(* CODESYS project safetymonitoring.library
   Author: Adam Garner
   Placeholder: SafetyMonitoring
   Title: SafetyMonitoring
   Version: 0.1.0.0
   Company: Ljmu

Project tree, tasks and I/O mapping:
  libraries: Tc2_Standard, * (Beckhoff Automation GmbH); Tc2_System, * (Beckhoff Automation GmbH); Tc3_Module, * (Beckhoff Automation GmbH)
  DUTs/
    data type e_EstopFBState
    data type e_EthercatCommError
    data type e_EthercatError
    data type e_EthercatState
    data type e_SafetyDiag
    data type e_SafetyGroupDiagnosis
    data type e_SafetyGroupState
    data type e_SafetyState
    data type ST_EL1918Inputs
    data type ST_EL1957Inputs
    data type ST_EL1957Outputs
    data type ST_EL2904Outputs
    data type ST_EstopFB
    data type ST_EstopFBDiag
    data type ST_EthercatStatus
    data type St_ModuleDescription
    data type ST_SafetyModule
    data type ST_SafetyStatus
    data type ST_WcStateStandard
  GVLs/
  POUs/
    function F_EthercatStateValid [ST]
    function block FB_EL1918Monitor [ST]: FB_init, GetInputs, SetInputs
    function block FB_EL1957Monitor [ST]
    function block FB_EL2904Monitor [ST]: FB_init
    function block FB_EstopFBCollectors [ST]: GetEstopData, MasterDataValid
    function block FB_EthercatModuleMonitor [ST]: CreateEthercatStatus, EtherCatStatusValid, FB_init, GetEthercatStatus, GetModuleDescription, LinkedOkVaild, ModuleDataValid, SetEthercatInputs, SetModuleDescription
    function block FB_SafetyEstopMonitor [ST]: FB_init, GetEstopName, GetEstopState, GetFlags, GetState, Reset, SetState
    function block FB_SafetyModuleCollector [ST]: GetSafetyStatus
    function block FB_SafetyModuleMonitor [ST]: CreateSafetyStatus, FB_init, GetSafetyStatus, SetSafetyInputs, ValidateSafetyStatus
    function block FB_SafetySystemMonitor [ST]: GetGlobalEstopStatus, SetMasterStatus
    interface ITF_SafetyModuleMonitor: CreateSafetyStatus, FB_init, GetEthercatStatus, GetModuleDescription, GetSafetyStatus, SetEthercatInputs, SetSafetyInputs, ValidateSafetyStatus
    program MAIN [ST]
  VISUs/
*)

// DUTs/e_EstopFBState
{attribute 'qualified_only'}
{attribute 'to_string'}
// Enum decribes states of a Estop function block 
TYPE e_EstopFBState :
(
	Undefined := 0,
	Run :=1,
	Stop:=2,
	Safe:=3,
	Error:=4,
	Reset:=5,
	Start:=6,
	Delayout:=8 
)BYTE;
END_TYPE
//source https://www.beckhoff.com/media/downloads/downloads/twinsafe-logic-fb-3.pdf PG50

// DUTs/e_EthercatCommError
{attribute 'qualified_only'}
{attribute 'to_string'}

TYPE e_EthercatCommError :
(	NoError:=0,
	InvalidError:=1,
	CommPortA := 16#1000,
	CommPortB := 16#2000,
	CommPortC := 16#4000,
	CommPortD := 16#8000
	
)UINT;
END_TYPE
// source https://infosys.beckhoff.com/english.php?content=../content/1033/b110_ethercat_optioninterface/1976021643.html&id=

// DUTs/e_EthercatError
{attribute 'qualified_only'}
{attribute 'to_string'}
// errors on a ethercat module 
TYPE e_EthercatError :
(
	NoError:=16#0000,
	SlaveSignalsError := 16#0010,
	InvalidProductCode := 16#0020,
	InitError := 16#0040,
	SlaveDisabled:= 16#0080,
	SlaveNotPresent :=16#0100,
	SlaveSignalLinkError := 16#0200,
	SlaveSignalMissingLink := 16#0400,
	SlaveSignalsUnexpectedLink := 16#0800,
	InvalidError:=5
	
)UINT;
END_TYPE
//source https://infosys.beckhoff.com/english.php?content=../content/1033/b110_ethercat_optioninterface/1976021643.html&id=

// DUTs/e_EthercatState
{attribute 'qualified_only'}
{attribute 'to_string'}
// the states of any ethercat module can be in 
TYPE e_EthercatState :
(
	InvalidState:=0,
	INIT := 1,
	PREOP :=2,
	BOOT :=3,
	SAFEOP:=4,
	OP :=8

)BYTE;
END_TYPE

//source https://infosys.beckhoff.com/english.php?content=../content/1033/b110_ethercat_optioninterface/1976021643.html&id=

// DUTs/e_SafetyDiag
{attribute 'qualified_only'}
{attribute 'to_string'}
//Enum descibes the final 4 bits of the Diagnostic varible that is common to all twinsafe modules 
TYPE e_SafetyDiag :
(	NoDiagnosisData:=0,
	InvalidCommand := 2#01,
	UnknownCommand := 2#10,
	InvalidConnectionID := 2#11,
	InvalidCRC := 2#100,
	WatchdogElapsed := 2#101,
	InvalidFSoEAddr := 2#110,
	InvalidData := 2#111,
	InvalidCommsParameterLength := 2#1000,
	InvalidCommsParameters := 2#1001,
	InvalidUserParametersLength := 2#1010,
	InvalidUserParameters := 2#1011,
	FSoEMasterReset := 2#1100,
	ModuleErrorOnSlaveComErrorActive := 2#1101,
	ModuleErrorOnSlaveErrAckActive := 2#1110,
	SlaveNotStartedOrUnexpectedErrorArgument :=2#1111
	
	
)USINT;
END_TYPE
// source https://download.beckhoff.com/download/Document/automation/twinsafe/TwinSAFE-Logic-FBen.pdf pg 20

// DUTs/e_SafetyGroupDiagnosis
{attribute 'qualified_only'}
TYPE e_SafetyGroupDiagnosis :
(
	NoError := 0,
	FBError:=1, 		//at least one FB is in ERROR state 
	ComError:=2, 		// at least one connection is faulty 
	ModuleError:=3, 	//the input ModuleFault is 1 
	CmpError:=4, 		//On startup, at least one analog FB input deviates from the last saved value (Power-On Analog Value Check Error) 
	DeativateError:=5, 	//The timeout has elapsed while waiting for the COM error in "passivate" mode of a manual control unit 
	RestartError :=6    //The TwinSAFE logic program was restarted because the EtherCAT connection was restarted or a user logged in without 
						//reloading the TwinSAFE logic program (or parts of it).
	
)USINT
;
END_TYPE
 // https://www.beckhoff.com/media/downloads/downloads/twinsafe-logic-fb-3.pdf pg 26

// DUTs/e_SafetyGroupState
{attribute 'qualified_only'}
TYPE e_SafetyGroupState :
(
	InvalidState:=0,
	Run:=1,				//Input RUN=1, no error in the group, and all connections have started up without error
	Stop:=2,			//Input RUN = 0 
	Error:=4,			//Group is in error, see Diagnostic information 
	Reset:=5,			//After a group error has occurred, all errors have been rectified and the Err Ack signal is 1 
	Start:=6,			// The group remains in this state as long as not all connections have started up after the start of the group (RUN=1) 
	StopError:=7,		// When the group is started or initialized, it assumes the STOPERROR status if the TwinSAFE connections are assigned to the group. 
						//The group switches from STOPERROR state into ERROR state if the Run input is TRUE. 
	Deactive:=16, 		//Group was deactivated via customizing
	WaitComError:=17 	// This state is set when the customizing function "Passivate" is selected and the system waits for ComError of the group
	
	
)USINT
;
END_TYPE
// source https://www.beckhoff.com/media/downloads/downloads/twinsafe-logic-fb-3.pdf pg26

// DUTs/e_SafetyState
{attribute 'qualified_only'}
{attribute 'to_string'}
//Enum descibes the State varible that is common to all twinsafe modules 
TYPE e_SafetyState :
(
	Reset := 100,
	Session:=101,
	Connection:=102,
	Parameter:=103,
	Data:=104,
	Shutdown:=105,
	ShutDownDeactivate:=106,
	StateDataNotAvailable:=0,
	InvalidState :=1
)USINT :=InvalidState
;
END_TYPE
// source https://download.beckhoff.com/download/Document/automation/twinsafe/TwinSAFE-Logic-FBen.pdf pg 21

// DUTs/ST_EL1918Inputs
// bit structure showing raw input state of a EL1918 module (8 channel safe inputs) should be mapped to the IO module 
TYPE ST_EL1918Inputs :
STRUCT
	Input1 :BIT;
	Input1Err :BIT;
	Input2 :BIT;
	Input2Err :BIT;
	Input3 :BIT;
	Input3Err :BIT;
	Input4 :BIT;
	Input4Err :BIT;
	Input5 :BIT;
	Input5Err :BIT;
	Input6 :BIT;
	Input6Err :BIT;
	Input7 :BIT;
	Input7Err :BIT;
	Input8 :BIT;
	Input8Err :BIT;
END_STRUCT
END_TYPE

// DUTs/ST_EL1957Inputs
// bit structure for all inputs of a E1957 8 channel safe input 4 safe outputs should be mapped to the IO 
TYPE ST_EL1957Inputs :
STRUCT
	Output1Err :BIT;// True if output 1 is in error state 
	Output2Err :BIT;
	Output3Err :BIT;
	Output4Err :BIT;
	Input1 :BIT;
	Input2 :BIT;
	Module1Err :BIT;//module 1 contains inputs 1 & 2 
	Input3 :BIT;
	Input4 :BIT;
	Module2Err :BIT;//module 2 contains inputs 3 & 4
	Input5 :BIT;
	Input6 :BIT;
	Module3Err :BIT;//module 3 contains inputs 5 & 6
	Input7 :BIT;
	Input8 :BIT;
	Module4Err :BIT;//module 4 contains inputs 7 & 8 
END_STRUCT
END_TYPE

// DUTs/ST_EL1957Outputs
TYPE ST_EL1957Outputs :
STRUCT
	Output1 :BIT;
	Output1ErrAck :BIT;
	Output2 :BIT;
	Output2ErrAck :BIT;
	Output3 :BIT;
	Output3ErrAck :BIT;
	Output4 :BIT;
	Output4ErrAck :BIT;
	InputModule1ErrAck :BIT;
	InputModule2ErrAck :BIT;
	InputModule3ErrAck :BIT;
	InputModule4ErrAck :BIT;
	
END_STRUCT
END_TYPE

// DUTs/ST_EL2904Outputs
TYPE ST_EL2904Outputs :
STRUCT
	Output1 :BIT;
	Output2 :BIT;
	Output3 :BIT;
	Output4 :BIT;
END_STRUCT
END_TYPE

// DUTs/ST_EstopFB
TYPE ST_EstopFB :
STRUCT
	EstopArea :STRING;
	State : e_EstopFBState;
	StrState: STRING;
	Diagnostics : ST_EstopFBDiag;
	Running :BOOL;
	Error:BOOL;
	Restart :BOOL;
END_STRUCT
END_TYPE

// DUTs/ST_EstopFBDiag
TYPE ST_EstopFBDiag :
STRUCT
	DiscrepancyErrInputGroup1 :BIT;
	DiscrepancyErrInputGroup2 :BIT;
	DiscrepancyErrInputGroup3 :BIT;
	DiscrepancyErrInputGroup4 :BIT;
	EDM1Err :BIT;
	EDM2Err :BIT;
	NA_1 :BIT;
	NA_2 :BIT;
	DiscErrInputGroup1 :BIT;
	DiscErrInputGroup2 :BIT;
	DiscErrInputGroup3 :BIT;
	DiscErrInputGroup4 :BIT;
	NA_3 :BIT;
	NA_4: BIT;
	NA_5: BIT;
	NA_6: BIT;
END_STRUCT
END_TYPE
// source https://www.beckhoff.com/media/downloads/downloads/twinsafe-logic-fb-3.pdf pg47

// DUTs/ST_EthercatStatus
// readable structure showing the status of any ethercat module 
TYPE ST_EthercatStatus :
STRUCT
	State :e_EthercatState;
	Error :e_EthercatError;
	CommError :e_EthercatCommError;
	DataValid:BOOL; // if false all data values from the module arent current 
	CablesOk:BOOL; // true if no comms error showing 
	LinkedOK :BOOL; // true if the values are linked to a module 
	ModuleOK:BOOL; // true is all values are normal excluding cables ok 
END_STRUCT
END_TYPE


// ethercat state definition https://infosys.beckhoff.com/english.php?content=../content/1033/tcsystemmanager/1089009035.html&id=4933952924797561914

// DUTs/St_ModuleDescription

//structure for storing data about the modules that are being monitored
TYPE St_ModuleDescription :
STRUCT
	ModuleName: STRING; // related to that it does 
	ModuleElectricalRef :STRING; // as shown on the wiring diagram
	ModuleAddress : INT; // termingal number shown in twincat 
	
END_STRUCT
END_TYPE

// DUTs/ST_SafetyModule
TYPE ST_SafetyModule :
STRUCT
	SafetyStatus : ST_SafetyStatus;
	strSafetyState :STRING;
	strSafetydiag :STRING;
	EthercatStatus : ST_EthercatStatus;
	strEthercatState : STRING;
	strEthercatError : STRING;
	strEthercatCommError : STRING;
	ModuleDescription : St_ModuleDescription; 
END_STRUCT
END_TYPE

// DUTs/ST_SafetyStatus
// readable structure for the current status of a safety module 
TYPE ST_SafetyStatus :
STRUCT
	State :e_SafetyState;
	Diagnosis : e_SafetyDiag;
	FSoESlaveError : BOOL;
	FSoESlaveFailSafeActive :BOOL;
	StartUp :BOOL;
	FSoEMasterFailSafeActive:BOOL;
	ModuleAllOk :BOOL; // summary ok flag 
END_STRUCT
END_TYPE

// source https://www.beckhoff.com/media/downloads/downloads/twinsafe-logic-fb-3.pdf pg47

// DUTs/ST_WcStateStandard
//structure for linking to a ethercat module 
TYPE ST_WcStateStandard :
STRUCT
	WcState :BIT :=TRUE; // 0 is datavalid
	InputToggle :BIT;	// toggles approx ever 1s 
END_STRUCT
END_TYPE

// POUs/F_EthercatStateValid
// checks for invalid ethercat states is used in the thercat module monitor can be changed to a internal fuction

FUNCTION F_EthercatStateValid : Bool
VAR_IN_OUT
	EthercatState : ST_EthercatStatus;
END_VAR
VAR
	// these arrays list all valid states so this code then loops through the states checks if its in the arrays 
	// so to add more states add to these arrays and increase the relevent for loop upper limit 
	EthercatStateValidValues : ARRAY [0..5] OF e_EthercatState:= [
								e_EthercatState.InvalidState,
								e_EthercatState.INIT,
								e_EthercatState.PREOP,
								e_EthercatState.BOOT,
								e_EthercatState.SAFEOP,
								e_EthercatState.OP];
	
	EthercatErrorValidValues : ARRAY [0..9] OF e_EthercatError := [
								e_EthercatError.NoError,
								e_EthercatError.SlaveSignalsError,
								e_EthercatError.InvalidProductCode,
								e_EthercatError.InitError,
								e_EthercatError.SlaveDisabled,
								e_EthercatError.SlaveNotPresent,
								e_EthercatError.SlaveSignalLinkError,
								e_EthercatError.SlaveSignalMissingLink,
								e_EthercatError.SlaveSignalsUnexpectedLink,
								e_EthercatError.InvalidError];	

EthercatCommErrorValidValues : ARRAY [0..5] OF e_EthercatCommError := [
								e_EthercatCommError.NoError,
								e_EthercatCommError.CommPortA,
								e_EthercatCommError.CommPortB,
								e_EthercatCommError.CommPortC,
								e_EthercatCommError.CommPortD];					
	State: INT;
	StateValid:BOOL:=FALSE;
	Error:INT;
	ErrorValid:BOOL:=FALSE;
	CommError:INT;
	CommErrorValid:BOOL:=FALSE;
	
END_VAR


FOR State := 0 TO 5 BY 1 DO
	IF (EthercatState.State = EthercatStateValidValues[state]) THEN
		StateValid:=TRUE;
	END_IF
END_FOR

IF NOT StateValid THEN
	EthercatState.State := e_EthercatState.InvalidState;
END_IF


FOR Error := 0 TO 9 BY 1 DO
	IF (EthercatState.Error = EthercatErrorValidValues[Error]) THEN
		ErrorValid:=TRUE;
	END_IF
END_FOR

IF NOT ErrorValid THEN
	EthercatState.Error := e_EthercatError.InvalidError;
END_IF

FOR CommError := 0 TO 5 BY 1 DO
	IF (EthercatState.CommError = EthercatCommErrorValidValues[CommError]) THEN
		CommErrorValid:=TRUE;
	END_IF
END_FOR

IF NOT CommErrorValid THEN
	EthercatState.CommError := e_EthercatCommError.InvalidError;
END_IF

F_EthercatStateValid := StateValid AND ErrorValid AND CommErrorValid;
//returns true if All values was valid

END_FUNCTION

// POUs/FB_EL1918Monitor
// used for a EL1918 addes inputs mapping and a okflag for the whole module and the inputs 
FUNCTION_BLOCK FB_EL1918Monitor EXTENDS FB_SafetyModuleMonitor
VAR
	ModuleInputs AT%I* :st_EL1918Inputs;
	InputsErrorFlag :BOOL; // False if any input has a error;
END_VAR

CreateSafetyStatus(inSafetyState:=SafetyState,inSafetyDiag:=SafetyDiagnosis,stSafetyStatusInOut:=stSafetyStatus);
CreateEthercatStatus(StateIn:= InputState,WCStateIn:= InputWcState,EthercatStatusOut=>stEthercatStatus);// main loop in here to be used in extended classes 
EthercatDatavalid:= EtherCatStatusValid(stEthercatStatusInOut:= stEthercatStatus);
LinkedOkVaild(TOFInOut:=LinkedOKTOF,InputToggleIn:= InputWcState.InputToggle,stEthercatStatusInOut:=stEthercatStatus);
ValidateSafetyStatus(stEthercatStateIn:= stEthercatStatus);// invalidate safety info if ethercat is down



IF ModuleInputs.Input1Err OR ModuleInputs.Input2Err
 OR ModuleInputs.Input3Err OR ModuleInputs.Input4Err
 OR ModuleInputs.Input5Err OR ModuleInputs.Input6Err 
 OR ModuleInputs.Input7Err  OR ModuleInputs.Input8Err THEN 
 InputsErrorFlag := FALSE ;

ELSE
	InputsErrorFlag := TRUE;
END_IF

METHOD FB_init : BOOL
VAR_INPUT
	bInitRetains : BOOL; // if TRUE, the retain variables are initialized (warm start / cold start)
	bInCopyCode : BOOL;  // if TRUE, the instance afterwards gets moved into the copy code (online change)
	NameIn: STRING;
	ElectricalRefIn :STRING;
	AddressIn : INT;
END_VAR
stModuleDescription.ModuleAddress := AddressIn;
stModuleDescription.ModuleElectricalRef:= ElectricalRefIn;
stModuleDescription.ModuleName:= NameIn;
END_METHOD

METHOD GetInputs
VAR_OUTPUT
	stInputsStatusOut : st_EL1918Inputs;
	OKFlagOut :bool;
END_VAR
stInputsStatusOut := ModuleInputs;
OkFlagOut := InputsErrorFlag;
END_METHOD

METHOD SetInputs : ST_SafetyStatus
VAR_INPUT
	Inputs : st_EL1918Inputs;
END_VAR
ModuleInputs := Inputs;
END_METHOD

END_FUNCTION_BLOCK

// POUs/MAIN
PROGRAM MAIN
VAR

END_VAR

END_PROGRAM

// POUs/FB_SafetyModuleMonitor
// this FB is used to monitor the State and Diagnosis of a safety module 
// includes a instance of a Ethercat module monitor this is so data is invalidated when ethercat network goes down  
FUNCTION_BLOCK FB_SafetyModuleMonitor EXTENDS FB_EthercatModuleMonitor IMPLEMENTS ITF_SafetyModuleMonitor
VAR
{attribute 'OPC.UA.DA' := '0'}
	SafetyState AT%I* :USINT; // should be linked to state in the process image inside the safety group controllers process image 
	{attribute 'OPC.UA.DA' := '0'}
	SafetyDiagnosis AT%I* :USINT;// should be linked to diag in the process image inside the safety group controllers process image 
	stSafetyStatus :ST_SafetyStatus ; // Structure containing process infomation
	// the init arguments are place holders its gets overwriten in this functions fb init 
	// the state and wcstate need mapping inside fbEthercatModuleMonitor

END_VAR

CreateSafetyStatus(inSafetyState:=SafetyState,inSafetyDiag:=SafetyDiagnosis,stSafetyStatusInOut:=stSafetyStatus);
CreateEthercatStatus(StateIn:= InputState,WCStateIn:= InputWcState,EthercatStatusOut=>stEthercatStatus);// main loop in here to be used in extended classes 
EthercatDatavalid:= EtherCatStatusValid(stEthercatStatusInOut:= stEthercatStatus);
LinkedOkVaild(TOFInOut:=LinkedOKTOF,InputToggleIn:= InputWcState.InputToggle,stEthercatStatusInOut:=stEthercatStatus);
ValidateSafetyStatus(stEthercatStateIn:= stEthercatStatus);// invalidate safety info if ethercat is down

// this takes in the state and diag and makes in ito the readable safety status structure see the st_safety structure definition for more details on the output
METHOD CreateSafetyStatus 
VAR_INPUT
inSafetyState :USINT;
inSafetyDiag  :USINT;
END_VAR
VAR_IN_OUT
	stSafetyStatusInOut : ST_SafetyStatus;
END_VAR
// check if State is in standard range if not invalidate state 
IF (inSafetyState=0) OR (inSafetyState=1) OR  ((inSafetyState<=107) AND (inSafetyState>=100)) THEN
stSafetyStatusInOut.State:=inSafetyState;
ELSE 
stSafetyStatusInOut.State:=e_SafetyState.InvalidState;
END_IF
// map the bools to the safety structure 
stSafetyStatusInOut.FSoEMasterFailSafeActive:=inSafetyDiag.7;
stSafetyStatusInOut.StartUp:= inSafetyDiag.6;
stSafetyStatusInOut.FSoESlaveFailSafeActive:=inSafetyDiag.5;
stSafetyStatusInOut.FSoESlaveError:=inSafetyDiag.4;
// final 4 bits make up the diagnosis 
stSafetyStatusInOut.Diagnosis:= inSafetyDiag AND 16#0F;

stSafetyStatusInOut.ModuleAllOk:= TRUE;
// checking if module is in an all ok state 
IF NOT (stSafetyStatusInOut.State = e_SafetyState.Data) THEN
stSafetyStatusInOut.ModuleAllOk:= FALSE;
END_IF

IF NOT stSafetyStatusInOut.Diagnosis = e_SafetyDiag.NoDiagnosisData THEN
	stSafetyStatusInOut.ModuleAllOk:= FALSE;
END_IF

IF NOT stSafetyStatusInOut.FSoESlaveError = FALSE THEN
	stSafetyStatusInOut.ModuleAllOk:= FALSE;
END_IF

IF NOT stSafetyStatusInOut.FSoESlaveFailSafeActive = FALSE THEN
	stSafetyStatusInOut.ModuleAllOk:= FALSE;
END_IF

IF NOT stSafetyStatusInOut.FSoEMasterFailSafeActive = FALSE THEN
	stSafetyStatusInOut.ModuleAllOk:= FALSE;
END_IF

IF NOT stSafetyStatusInOut.StartUp = FALSE THEN
	stSafetyStatusInOut.ModuleAllOk:= FALSE;
END_IF
END_METHOD

// the input arguments are to fill out the module description structure in the ethercat module fb
METHOD FB_init : BOOL
VAR_INPUT
	bInitRetains : BOOL; // if TRUE, the retain variables are initialized (warm start / cold start)
	bInCopyCode : BOOL;  // if TRUE, the instance afterwards gets moved into the copy code (online change)
	NameIn: STRING;
	ElectricalRefIn :STRING;
	AddressIn : INT;
END_VAR
stModuleDescription.ModuleAddress := AddressIn;
stModuleDescription.ModuleElectricalRef:= ElectricalRefIn;
stModuleDescription.ModuleName:= NameIn;
END_METHOD


METHOD GetSafetyStatus : ST_SafetyStatus
VAR_OUTPUT
	stSafetyStatusOut : ST_SafetyStatus;
END_VAR
stSafetyStatusOut :=stSafetyStatus;
END_METHOD

// mostly used in unit testing as it allows inputs to the Safety module without linked varibles 
METHOD SetSafetyInputs
VAR_INPUT
	StateIn  :USINT;
	DiagnosisIn  :USINT;
END_VAR
SafetyState:=StateIn;
SafetyDiagnosis :=DiagnosisIn;
END_METHOD

// invalidates safety structure when data isnt valid is called from this functions main 
METHOD ValidateSafetyStatus
VAR_INPUT
	stEthercatStateIn: ST_EthercatStatus;
END_VAR

IF NOT stEthercatStateIn.DataValid THEN
	stSafetyStatus.State := e_SafetyState.StateDataNotAvailable;
	stSafetyStatus.Diagnosis := e_SafetyDiag.WatchdogElapsed;
	stSafetyStatus.FSoESlaveError:= TRUE;
	stSafetyStatus.FSoESlaveFailSafeActive:= TRUE;
	stSafetyStatus.StartUp:= TRUE;
	stSafetyStatus.FSoEMasterFailSafeActive:= TRUE;
	stSafetyStatus.ModuleAllOk := FALSE;
END_IF
END_METHOD

END_FUNCTION_BLOCK

// POUs/FB_EthercatModuleMonitor
//this fb is to be used on every ethercat module with the InputState mapped to State  and inputWCStates mapped to  Wcstate and input toggle 
// this gives you a structure with the status on the module in a readable format and some useful summary booleans 
// the fb init is used to fill out module infomation this will later be used in events and lets you track down faulty modules quickly 
FUNCTION_BLOCK FB_EthercatModuleMonitor
VAR

	InputState AT%I*	:UINT;	// link to ethercat state in process image 
	InputWcState AT%I* : ST_WcStateStandard; // structure including wc state and input toggle to be linked to process image 
	stEthercatStatus : ST_EthercatStatus; // output summary structure 
	stModuleDescription: ST_ModuleDescription; 
	EthercatDatavalid :BOOL;
	LinkedOKTOF :TOF := (IN :=True,PT:= t#2s);
END_VAR

CreateEthercatStatus(StateIn:= InputState,WCStateIn:= InputWcState,EthercatStatusOut=>stEthercatStatus);// main loop in here to be used in extended classes 
EthercatDatavalid:= EtherCatStatusValid(stEthercatStatusInOut:= stEthercatStatus);
LinkedOkVaild(TOFInOut:=LinkedOKTOF,InputToggleIn:= InputWcState.InputToggle,stEthercatStatusInOut:=stEthercatStatus);

METHOD PROTECTED CreateEthercatStatus
VAR_INPUT
	StateIn :UINT;
	WCStateIn: ST_WcStateStandard;
END_VAR

VAR_OUTPUT
	EthercatStatusOut : ST_EthercatStatus;
	
END_VAR
// split date into the components for info is found in the ST_EthercatState definition of what this includes 
EthercatStatusOut.State := UINT_TO_BYTE(InputState AND 16#000F);
EthercatStatusOut.Error := InputState AND 16#0FF0;
EthercatStatusOut.CommError := InputState AND 16#F000;

EthercatStatusOut.DataValid:= NOT InputWcState.WcState; // Wcstate 0 means data valid 


//cables ok check 
	EthercatStatusOut.CablesOk:= FALSE;
IF (EthercatStatusOut.CommError = e_EthercatCommError.NoError) THEN
	EthercatStatusOut.CablesOk:= TRUE;
END_IF
END_METHOD

// internal function to check for Validity on the EthercatStatus
METHOD PROTECTED EtherCatStatusValid : BOOL
VAR_IN_OUT
	stEthercatStatusInOut : ST_EthercatStatus;
END_VAR
VAR
	// these arrays list all valid states so this code then loops through the states checks if its in the arrays 
	// so to add more states add to these arrays and increase the relevent for loop upper limit 
	EthercatStatusValidValues : ARRAY [0..5] OF e_EthercatState:= [
								e_EthercatState.InvalidState,
								e_EthercatState.INIT,
								e_EthercatState.PREOP,
								e_EthercatState.BOOT,
								e_EthercatState.SAFEOP,
								e_EthercatState.OP];
	
	EthercatErrorValidValues : ARRAY [0..9] OF e_EthercatError := [
								e_EthercatError.NoError,
								e_EthercatError.SlaveSignalsError,
								e_EthercatError.InvalidProductCode,
								e_EthercatError.InitError,
								e_EthercatError.SlaveDisabled,
								e_EthercatError.SlaveNotPresent,
								e_EthercatError.SlaveSignalLinkError,
								e_EthercatError.SlaveSignalMissingLink,
								e_EthercatError.SlaveSignalsUnexpectedLink,
								e_EthercatError.InvalidError];	

EthercatCommErrorValidValues : ARRAY [0..5] OF e_EthercatCommError := [
								e_EthercatCommError.NoError,
								e_EthercatCommError.CommPortA,
								e_EthercatCommError.CommPortB,
								e_EthercatCommError.CommPortC,
								e_EthercatCommError.CommPortD];
					
	State: INT;
	StateValid:BOOL:=FALSE;
	Error:INT;
	ErrorValid:BOOL:=FALSE;
	CommError:INT;
	CommErrorValid:BOOL:=FALSE;
	
END_VAR
FOR State := 0 TO 5 BY 1 DO
	IF (stEthercatStatusInOut.State = EthercatStatusValidValues[state]) THEN
		StateValid:=TRUE;
	END_IF
END_FOR

IF NOT StateValid THEN
	stEthercatStatusInOut.State := e_EthercatState.InvalidState;
END_IF


FOR Error := 0 TO 9 BY 1 DO
	IF (stEthercatStatusInOut.Error = EthercatErrorValidValues[Error]) THEN
		ErrorValid:=TRUE;
	END_IF
END_FOR

IF NOT ErrorValid THEN
	stEthercatStatusInOut.Error := e_EthercatError.InvalidError;
END_IF

FOR CommError := 0 TO 5 BY 1 DO
	IF (stEthercatStatusInOut.CommError = EthercatCommErrorValidValues[CommError]) THEN
		CommErrorValid:=TRUE;
	END_IF
END_FOR

IF NOT CommErrorValid THEN
	stEthercatStatusInOut.CommError := e_EthercatCommError.InvalidError;
END_IF

EtherCatStatusValid := StateValid AND ErrorValid AND CommErrorValid;
//returns true if All values was valid
END_METHOD

// arguments are used to fill module description structure 

METHOD FB_init : BOOL
VAR_INPUT
	bInitRetains : BOOL; // if TRUE, the retain variables are initialized (warm start / cold start)
	bInCopyCode : BOOL;  // if TRUE, the instance afterwards gets moved into the copy code (online change)
	NameIn: STRING;
	ElectricalRefIn :STRING;
	AddressIn : INT;
END_VAR
stModuleDescription.ModuleAddress := AddressIn;
stModuleDescription.ModuleElectricalRef:= ElectricalRefIn;
stModuleDescription.ModuleName:= NameIn;
END_METHOD

METHOD PUBLIC  GetEthercatStatus 
VAR_OUTPUT
	stEthercatStatusOut: ST_EthercatStatus;
END_VAR
stEthercatStatusOut := stEthercatStatus;
END_METHOD

METHOD PUBLIC GetModuleDescription 
VAR_OUTPUT
	stDescriptionOut :St_ModuleDescription;
END_VAR
stDescriptionOut:=stModuleDescription;
END_METHOD

METHOD PROTECTED LinkedOkVaild
VAR_INPUT
	InputToggleIn :BOOL;
END_VAR
VAR_IN_OUT
	TOFInOut :TOF;
	stEthercatStatusInOut :ST_EthercatStatus;
END_VAR

VAR


END_VAR
// linked ok check 


TOFInOut(IN:=InputToggleIn,Q=>stEthercatStatusInOut.LinkedOK);
// if not linked corrected invalidate data 
IF NOT stEthercatStatusInOut.LinkedOK THEN
	stEthercatStatusInOut.DataValid:=FALSE;	
END_IF

// all ok Check 
stEthercatStatusInOut.ModuleOk:= FALSE;
IF stEthercatStatusInOut.DataValid AND stEthercatStatusInOut.LinkedOK AND (stEthercatStatusInOut.State=e_EthercatState.OP) THEN
	stEthercatStatusInOut.ModuleOk := TRUE;
END_IF
END_METHOD

// fuction can be used if you need a simple validity check on data out of a module 
METHOD PUBLIC ModuleDataValid :BOOL
VAR_OUTPUT
	
END_VAR
ModuleDataValid := stEthercatStatus.DataValid;
END_METHOD

// only use if not varibles linked such as in unit testing 
METHOD Public SetEthercatInputs
VAR_INPUT
	StateIn :UINT;	
	WcStateIn : ST_WcStateStandard;
END_VAR
InputState:=StateIn;
InputWcState:= WcStateIn;
END_METHOD

// this is set in the fb init so use only if changing the structure 
METHOD INTERNAL SetModuleDescription :BOOL
VAR_INPUT
	DescriptionIn : St_ModuleDescription;
END_VAR
stModuleDescription:=DescriptionIn;
END_METHOD

END_FUNCTION_BLOCK

// POUs/ITF_SafetyModuleMonitor
INTERFACE ITF_SafetyModuleMonitor

METHOD CreateSafetyStatus
VAR_INPUT
inSafetyState :USINT;
inSafetyDiag  :USINT;
END_VAR
VAR_IN_OUT
	stSafetyStatusInOut : ST_SafetyStatus;
END_VAR
END_METHOD

METHOD FB_init : BOOL
VAR_INPUT
	bInitRetains : BOOL; // if TRUE, the retain variables are initialized (warm start / cold start)
	bInCopyCode : BOOL;  // if TRUE, the instance afterwards gets moved into the copy code (online change)
	NameIn: STRING;
	ElectricalRefIn :STRING;
	AddressIn : INT;
END_VAR
END_METHOD

METHOD GetEthercatStatus 
VAR_OUTPUT
	stEthercatStatusOut : ST_EthercatStatus;
END_VAR
END_METHOD

METHOD GetModuleDescription 
VAR_OUTPUT
	stDescriptionOut : St_ModuleDescription;
END_VAR
END_METHOD

METHOD GetSafetyStatus  : ST_SafetyStatus
VAR_OUTPUT
	stSafetyStatusOut : ST_SafetyStatus;
END_VAR
END_METHOD

METHOD SetEthercatInputs 
VAR_INPUT
	StateIn :UINT;	
	WcStateIn : ST_WcStateStandard;
END_VAR
END_METHOD

METHOD SetSafetyInputs 
VAR_INPUT
	StateIn  :USINT;
	DiagnosisIn  :USINT;
END_VAR
END_METHOD

METHOD ValidateSafetyStatus 
VAR_INPUT
	stEthercatStateIn: ST_EthercatStatus;
END_VAR
END_METHOD

END_INTERFACE

// POUs/FB_EL1957Monitor
FUNCTION_BLOCK FB_EL1957Monitor
VAR
	State AT%I* :USINT;
	Diag AT%I* :USINT;
	Status :ST_SafetyStatus;
	Outputs AT%I* :ST_EL2904Outputs;
	Inputs AT%I* :ST_EL1957Inputs;
END_VAR

// no yet implemented

END_FUNCTION_BLOCK

// POUs/FB_EL2904Monitor
// fb is used for EL2904 modules adds the outputs into the module 

FUNCTION_BLOCK FB_EL2904Monitor EXTENDS FB_SafetyModuleMonitor
VAR
	Outputs AT%I* :ST_EL2904Outputs;
END_VAR

CreateSafetyStatus(inSafetyState:=SafetyState,inSafetyDiag:=SafetyDiagnosis,stSafetyStatusInOut:=stSafetyStatus);
CreateEthercatStatus(StateIn:= InputState,WCStateIn:= InputWcState,EthercatStatusOut=>stEthercatStatus);// main loop in here to be used in extended classes 
EthercatDatavalid:= EtherCatStatusValid(stEthercatStatusInOut:= stEthercatStatus);
LinkedOkVaild(TOFInOut:=LinkedOKTOF,InputToggleIn:= InputWcState.InputToggle,stEthercatStatusInOut:=stEthercatStatus);
ValidateSafetyStatus(stEthercatStateIn:= stEthercatStatus);// invalidate safety info if ethercat is down

METHOD FB_init : BOOL
VAR_INPUT
	bInitRetains : BOOL; // if TRUE, the retain variables are initialized (warm start / cold start)
	bInCopyCode : BOOL;  // if TRUE, the instance afterwards gets moved into the copy code (online change)
	NameIn: STRING;
	ElectricalRefIn :STRING;
	AddressIn : INT;
END_VAR
stModuleDescription.ModuleAddress := AddressIn;
stModuleDescription.ModuleElectricalRef:= ElectricalRefIn;
stModuleDescription.ModuleName:= NameIn;
END_METHOD

END_FUNCTION_BLOCK

// POUs/FB_EstopFBCollectors
FUNCTION_BLOCK FB_EstopFBCollectors
VAR_IN_OUT
	stEstopArrayInOut :ARRAY [*] OF ST_estopFB;
END_VAR
VAR_INPUT
	EstopArraySizeIn: UINT;
END_VAR
VAR
		Estop :UINT;
		DataValid:BOOL:= FALSE;  // if not wrote to data is invalid
		stDiagnostic: ST_EstopFBDiag;
END_VAR

FOR Estop :=0 TO EstopArraySizeIn BY 1 DO 

	IF NOT DataValid THEN
		stEstopArrayInOut[Estop].Diagnostics:=stDiagnostic;
		stEstopArrayInOut[Estop].Error:= TRUE;
		stEstopArrayInOut[Estop].Running:=FALSE;
		stEstopArrayInOut[Estop].State:=e_EstopFBState.Undefined;	
	END_IF
	stEstopArrayInOut[Estop].StrState:=TO_STRING(stEstopArrayInOut[Estop].State);
END_FOR

METHOD GetEstopData : BOOL
VAR_INPUT
	SafetyEstopRefIn : REFERENCE TO FB_SafetyEstopMonitor;
	EstopIndexIn:UINT;
	EstopArraySizeIn:UINT;
END_VAR
VAR_IN_OUT
	stEstopArrayInOut :ARRAY [*] OF ST_estopFB;
END_VAR
VAR
	stDiagnostic: ST_EstopFBDiag;
	eState: e_EstopFBState;
	RunningFlag: BOOL;
	ErrorFlag: BOOL;
	EstopArea: STRING;
END_VAR
GetEstopData:=TRUE;

IF __ISVALIDREF(SafetyEstopRefIn) AND EstopIndexIn<=EstopArraySizeIn THEN // checking function pointer is valid and the array index is in range 
	SafetyEstopRefIn.GetState(stDiagnosticOut=>stDiagnostic,eStateOut=>eState);
	SafetyEstopRefIn.GetFlags(RunningFlagOut=>RunningFlag,ErrorFlagOut=>ErrorFlag);
	SafetyEstopRefIn.GetEstopName(NameOut=>EstopArea);
	//InputReference.Reset(Enable := EstopAreas[EstopNumber].Restart); crashes plc needs investigating 
	GetEstopData:= FALSE;
END_IF

IF EstopIndexIn<=EstopArraySizeIn THEN
	stEstopArrayInOut[EstopIndexIn].Diagnostics:=stDiagnostic;
	stEstopArrayInOut[EstopIndexIn].Error:= ErrorFlag;
	stEstopArrayInOut[EstopIndexIn].Running:=RunningFlag;
	stEstopArrayInOut[EstopIndexIn].State:=eState;
	stEstopArrayInOut[EstopIndexIn].EstopArea:= EstopArea;
		GetEstopData:= FALSE;
END_IF
END_METHOD

METHOD PUBLIC MasterDataValid
VAR_INPUT
	DataValidIn :BOOL;
END_VAR
DataValid := DataValidIn;
END_METHOD

END_FUNCTION_BLOCK

// POUs/FB_SafetyEstopMonitor
// this FB is to monitor the Estop twinsafe FB and structure the data rawstate and diagnostic are the inputs 
FUNCTION_BLOCK FB_SafetyEstopMonitor
VAR
	{attribute 'OPC.UA.DA' := '0'}
	InputEstopState AT%I* :USINT;  // map to state and diag of this fb found under the master in IO 
	{attribute 'OPC.UA.DA' := '0'}
	bitStEstopDiagnostic AT%I* :ST_EstopFBDiag;
	eEstopState :e_EstopFBState;
	Running :BOOL:=False; // safety block is running 
	Error :BOOL;
	Restart AT%Q*:BOOL; // bool to reset FB link to function block Restart not implemented
	AreaName :STRING;
END_VAR

eEstopState:=InputEstopState;
// check if invalid state only 8 possible states so check if in range 
IF (eEstopState>8) THEN
	eEstopState := e_EstopFBState.Undefined;
END_IF
// set running flag 
IF (eEstopState =e_EstopFBState.Run) THEN
	Running := TRUE;
ELSE 
	Running := FALSE;
END_IF
// set error flag 
IF (eEstopState =e_EstopFBState.Error) OR (eEstopState =e_EstopFBState.Undefined)  THEN
	Error := TRUE;
ELSE
	Error := FALSE;
END_IF

METHOD FB_init : BOOL
VAR_INPUT
	bInitRetains : BOOL; // if TRUE, the retain variables are initialized (warm start / cold start)
	bInCopyCode : BOOL;  // if TRUE, the instance afterwards gets moved into the copy code (online change)
	NameIn :string;
END_VAR
AreaName := NameIn ;
END_METHOD

METHOD GetEstopName
VAR_OUTPUT
	NameOut :string;
END_VAR
NameOut := areaName;
END_METHOD

// returns a Bool False if Estop Block is running with no faults otherwise True
METHOD GetEstopState : BOOL
VAR
END_VAR
IF Running THEN
	GetEstopState:= FALSE; 

ELSE
	GetEstopState:=TRUE;
END_IF
END_METHOD

METHOD GetFlags
VAR_OUTPUT
	RunningFlagOut :BOOL;
	ErrorFlagOut:BOOL;
END_VAR
RunningFlagOut :=Running;
ErrorFlagOut := Error;
END_METHOD

// returns the structured fb status and Diagnostics 
METHOD GetState
VAR_OUTPUT
	stDiagnosticOut  :ST_EstopFBDiag;
	eStateOut :e_EstopFBState;
END_VAR
stDiagnosticOut := bitStEstopDiagnostic;
eStateOut := eEstopState;
END_METHOD

// Enable with reset back to false after one cycle 
METHOD Reset : BOOL
VAR_IN_OUT
	EnableInOut :BOOL;
END_VAR
IF EnableInOut THEN
EnableInOut := FALSE;
Restart:= TRUE;
ELSE
Restart:=FALSE;	

END_IF
END_METHOD

//function used if varibles arent linked directly in FB 
// also useful for unit testing
METHOD PUBLIC SetState
VAR_INPUT
	StateIn :USINT;
	DiagnosticIn  :ST_EstopFBDiag;
END_VAR
InputEstopState := StateIn;
bitStEstopDiagnostic := DiagnosticIn;
END_METHOD

END_FUNCTION_BLOCK

// POUs/FB_SafetyModuleCollector
FUNCTION_BLOCK FB_SafetyModuleCollector
VAR_IN_OUT
	stModuleArrayInOut :ARRAY [*] OF ST_SafetyModule;
END_VAR
VAR_INPUT
ModuleArraySizeIn: UINT;
END_VAR
VAR_TEMP
	Module :uint;
END_VAR

FOR Module := 0 TO ModuleArraySizeIn BY 1 DO
	stModuleArrayInOut[Module].strSafetyState:= TO_STRING(stModuleArrayInOut[Module].SafetyStatus.State);
	stModuleArrayInOut[Module].strSafetyDiag:= TO_STRING(stModuleArrayInOut[Module].SafetyStatus.Diagnosis);
	stModuleArrayInOut[Module].strEthercatState:= TO_STRING(stModuleArrayInOut[Module].EthercatStatus.State);
	stModuleArrayInOut[Module].strEthercatError:= TO_STRING(stModuleArrayInOut[Module].EthercatStatus.Error);
	stModuleArrayInOut[Module].strEthercatCommError:= TO_STRING(stModuleArrayInOut[Module].EthercatStatus.CommError);
END_FOR

METHOD GetSafetyStatus : BOOL
VAR_INPUT
	SafetyModuleRefIn : REFERENCE TO FB_SafetyModuleMonitor;
	ModuleIndexIn :UINT;
	ModuleArraySizeIn :UINT;
//inputSafetyStatus : ST_SafetyStatus;
END_VAR
VAR_IN_OUT
	StModuleArrayInOut :ARRAY [*] OF ST_SafetyModule;
END_VAR
	
VAR
	
	stSafetyStatus: ST_SafetyStatus;
	stEthercatStatus : ST_EthercatStatus;
	stModuleDescription : St_ModuleDescription;
END_VAR
GetSafetyStatus:= TRUE;
IF __ISVALIDREF(SafetyModuleRefIn) THEN
SafetyModuleRefIn.GetSafetyStatus(stSafetyStatusOut=> stSafetyStatus);
SafetyModuleRefIn.GetEthercatStatus(stEthercatStatusOut=> stEthercatStatus);
SafetyModuleRefIn.GetModuleDescription(stDescriptionOut=> stModuleDescription);
GetSafetyStatus:= FALSE;
END_IF

IF ModuleIndexIn <= ModuleArraySizeIn THEN
StModuleArrayInOut[ModuleIndexIn].SafetyStatus:= stSafetyStatus;
StModuleArrayInOut[ModuleIndexIn].EthercatStatus:= stEthercatStatus;
StModuleArrayInOut[ModuleIndexIn].ModuleDescription := stModuleDescription;
GetSafetyStatus:=FALSE;
END_IF
END_METHOD

END_FUNCTION_BLOCK

// POUs/FB_SafetySystemMonitor
/// this FB is used to monitor the State and Diagnosis of the Whole Safety System 
FUNCTION_BLOCK FB_SafetySystemMonitor
VAR
	Run AT%Q*:BOOL:=TRUE;
	ErrAck AT%Q* :BOOL;
	eSafetyGroupState AT%I* :e_SafetyGroupState;
	eSafetyGroupDiagnosis AT%I* :e_SafetyGroupDiagnosis;
	stEthercatStatus :ST_EthercatStatus;
	GlobalEstopStatus AT%I* :BOOL :=FALSE; // true is system Running false is system Activated(tripped)
	
END_VAR

IF NOT  stEthercatStatus.DataValid THEN
	eSafetyGroupState := e_SafetyGroupState.Error;
	eSafetyGroupDiagnosis := e_SafetyGroupDiagnosis.ComError;
	GlobalEstopStatus:= FALSE;
END_IF

// returns a boolean true if system is running false is system has activated(tripped) 
METHOD PUBLIC GetGlobalEstopStatus : BOOL
VAR_INPUT
END_VAR
GetGlobalEstopStatus:= GlobalEstopStatus;
END_METHOD

METHOD PUBLIC SetMasterStatus
VAR_INPUT
	StEthercatStatusIn :ST_EthercatStatus;
END_VAR
stEthercatStatus:= StEthercatStatusIn;
END_METHOD

END_FUNCTION_BLOCK
